(* CODESYS project Pistons innlevering 4 Biraveen.export

Project tree, tasks and I/O mapping:
  Device : CODESYS Control Win V3 x64, 3S - Smart Software Solutions GmbH, version 3.5.16.30
    application Application
      libraries: Standard, * (System)
      task MainTask (cyclic, interval 100 ms, priority 1) calls PLC_PRG
      task VISU_TASK (cyclic, interval 100 ms, priority 31) calls VisuElems.Visu_Prg
      global variables GVL
      function block egendefinert_ANDport [ST]
      function block Pistons [ST]
      program PLC_PRG [CFC]
      function block POU [ST]
      function block POU_1 [ST]
      function block seq4 [ST]
      function block Seq_1 [ST]
      visualisation Visualization
*)

// Device/Application/GVL
{attribute 'qualified_only'}
VAR_GLOBAL
	Piston1_IN: BOOL;
	Piston1_OUT: BOOL;
	Piston2_IN: BOOL;
	Piston2_OUT: BOOL;
	Piston3_IN: BOOL;
	Piston3_OUT: BOOL;
	Piston4_IN: BOOL;
	Piston4_OUT: BOOL;
END_VAR

// Device/Application/PLC_PRG
PROGRAM PLC_PRG
VAR
	Pistons_1: Pistons;
	RESET_0: POU; // første sekvens
	Start_knapp: BOOL;
	ElapsedTIme: TIME;
	TON_0: TON;
	DELAY_1: TON;
	Seq_1_0: Seq_1; // andre sekvens
	Delay_2: TON;
	seq_2: POU_1; // tredje sekvens
	Delay_3: TON;
	Seq_3: seq4; //dette er fjerde sekvens
	Delay_4: TON;
	port: egendefinert_ANDport; // egt en OR port-ish!!
	Delay_5: TON; // RESET delayen
END_VAR

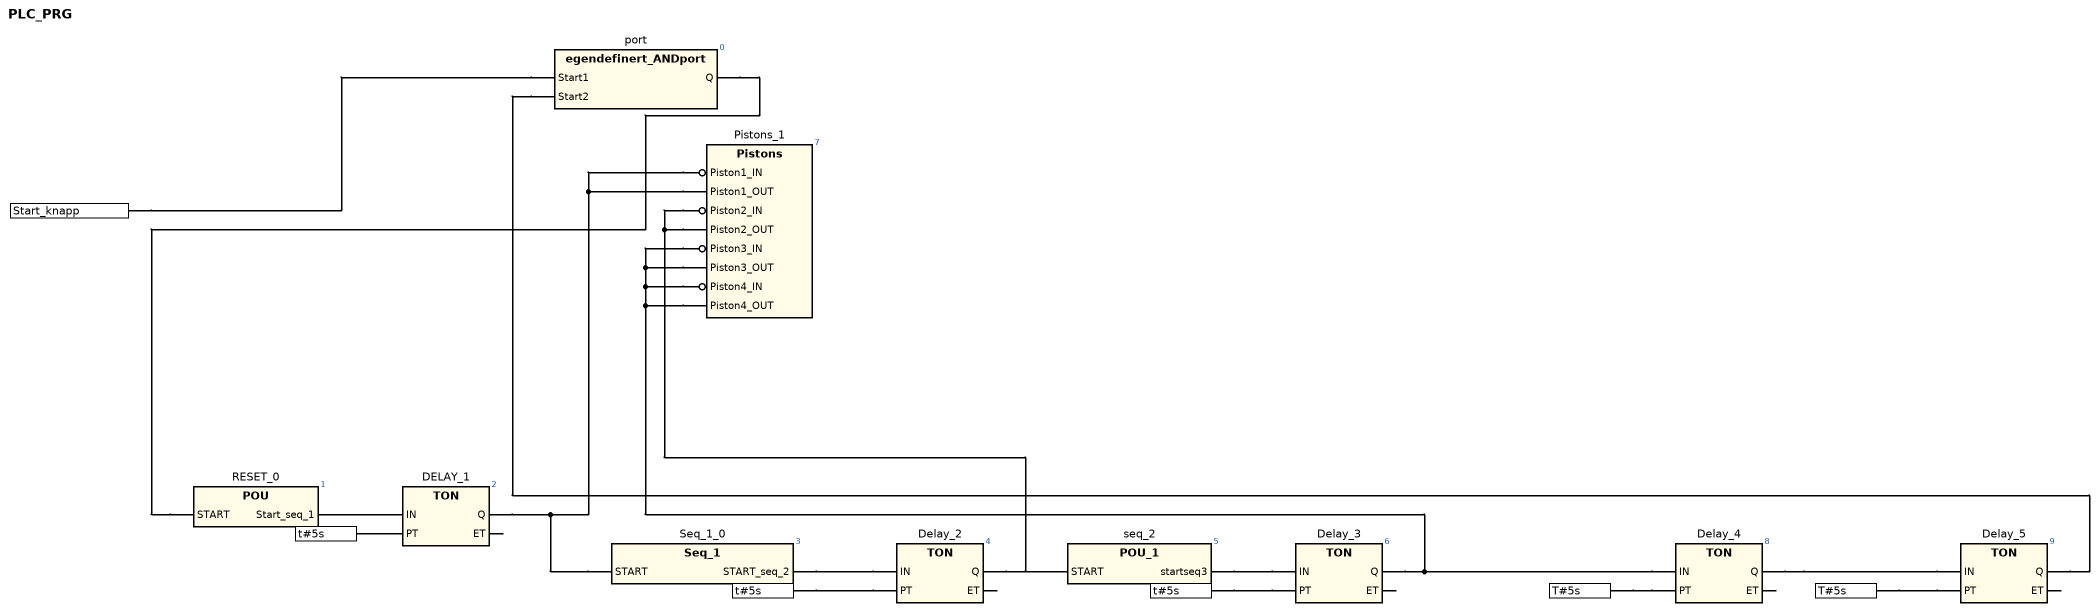
port(Start1 := Start_knapp, Start2 := Delay_5.Q); // egendefinert_ANDport
RESET_0(START := port.Q); // POU
DELAY_1(IN := RESET_0.Start_seq_1, PT := t#5s); // TON
Seq_1_0(START := DELAY_1.Q); // Seq_1
Delay_2(IN := Seq_1_0.START_seq_2, PT := t#5s); // TON
seq_2(START := Delay_2.Q); // POU_1
Delay_3(IN := seq_2.startseq3, PT := t#5s); // TON
Pistons_1(
    Piston1_IN := NOT DELAY_1.Q,
    Piston1_OUT := DELAY_1.Q,
    Piston2_IN := NOT Delay_2.Q,
    Piston2_OUT := Delay_2.Q,
    Piston3_IN := NOT Delay_3.Q,
    Piston3_OUT := Delay_3.Q,
    Piston4_IN := NOT Delay_3.Q,
    Piston4_OUT := Delay_3.Q); // Pistons
Delay_4(IN := Delay_3.Q, PT := T#5s); // TON
Delay_5(IN := Delay_4.Q, PT := T#5s); // TON

END_PROGRAM

// Device/Application/Pistons
FUNCTION_BLOCK Pistons
VAR_INPUT
	Piston1_IN : BOOL := FALSE;
	Piston1_OUT : BOOL := FALSE;
	Piston2_IN : BOOL := FALSE;
	Piston2_OUT : BOOL := FALSE;
	Piston3_IN : BOOL := FALSE;
	Piston3_OUT : BOOL := FALSE;
	Piston4_IN : BOOL := FALSE;
	Piston4_OUT : BOOL := FALSE;

END_VAR
VAR_OUTPUT
END_VAR
VAR
	Hide_Piston_1 : BOOL := TRUE;
	Hide_Piston_2 : BOOL := TRUE;
	Hide_Piston_3 : BOOL := TRUE;
	Hide_Piston_4 : BOOL := TRUE;
	Reset : BOOL := FALSE;
	Start: BOOL;
	Variabel_1: REAL;
	Tstart1 : TIME;
	variabel: REAL;
END_VAR

IF NOT Reset THEN
	
	IF Piston1_OUT AND NOT Piston1_IN THEN 
		Hide_Piston_1 := FALSE;
	ELSIF Piston1_IN AND NOT Piston1_OUT THEN
		Hide_Piston_1 := TRUE;
	ELSE
		Hide_Piston_1 := Hide_Piston_1;
	END_IF

	IF Piston2_OUT AND NOT Piston2_IN THEN
		Hide_Piston_2 := FALSE;
	ELSIF Piston2_IN AND NOT Piston2_OUT THEN
		Hide_Piston_2 := TRUE;
	ELSE
		Hide_Piston_2 := Hide_Piston_2;
	END_IF

	IF Piston3_OUT AND NOT Piston3_IN THEN
		Hide_Piston_3 := FALSE;
	ELSIF Piston3_IN AND NOT Piston3_OUT THEN
		Hide_Piston_3 := TRUE;
	ELSE
		Hide_Piston_3 := Hide_Piston_3;
	END_IF
	
	IF Piston4_OUT AND NOT Piston4_IN THEN
		Hide_Piston_4 := FALSE;
	ELSIF Piston4_IN AND NOT Piston4_OUT THEN
		Hide_Piston_4 := TRUE;
	ELSE
		Hide_Piston_4 := Hide_Piston_4;
	END_IF

ELSE
	Hide_Piston_1 := TRUE;
	Hide_Piston_2 := TRUE;
	Hide_Piston_3 := TRUE;
	Hide_Piston_4 := TRUE;
	Piston1_IN := FALSE;
	Piston1_OUT := FALSE;
	Piston2_IN := FALSE;
	Piston2_OUT := FALSE;
	Piston3_IN := FALSE;
	Piston3_OUT := FALSE;
	Piston4_IN := FALSE;
	Piston4_OUT := FALSE;
	variabel := 0;
END_IF

IF Hide_piston_2 = FALSE AND variabel = 0  THEN 
	HIDE_Piston_1 := TRUE;
END_IF

IF Hide_piston_3 = FALSE THEN 
	HIDE_Piston_2 := TRUE;
END_IF

//IF Hide_piston_4 = FALSE THEN 
	//HIDE_Piston_3 := TRUE;
	//variabel := 1;
//END_IF

// IF Hide_piston_4 = FALSE AND variabel = 1 THEN 
	//HIDE_Piston_1 := TRUE;
	//variabel := 0;
//END_IF

END_FUNCTION_BLOCK

// Device/Application/egendefinert_ANDport
FUNCTION_BLOCK egendefinert_ANDport
VAR_INPUT
	Start1 : BOOL;
	Start2 : BOOL;
END_VAR
VAR_OUTPUT
END_VAR
VAR
	Q : BOOL;
END_VAR

IF Start1 = FALSE AND Start2 = FALSE THEN
	Q := FALSE; 
END_IF

IF Start1 = TRUE AND Start2 = FALSE THEN
	Q := TRUE; 
END_IF

IF Start1 = FALSE AND Start2 = TRUE THEN
	Q := TRUE; 
END_IF

IF Start1 = TRUE AND Start2 = TRUE THEN
	Q := FALSE; 
END_IF

IF Q = FALSE AND START2 = TRUE THEN
	Q := TRUE; 
END_IF

END_FUNCTION_BLOCK

// Device/Application/POU_1
FUNCTION_BLOCK POU_1
VAR_INPUT
	START : BOOL;
END_VAR
VAR_OUTPUT
END_VAR
VAR
	Startseq3 : BOOL;
END_VAR

IF START = TRUE THEN 
	STARTseq3 := TRUE;
END_IF

IF START = FALSE THEN 
	STARTseq3 := FALSE;
END_IF

END_FUNCTION_BLOCK

// Device/Application/POU
FUNCTION_BLOCK POU
VAR_INPUT
	START : BOOL;
END_VAR
VAR_OUTPUT

END_VAR
VAR
	Start_seq_1: BOOL;
	pistonin : BOOL;
	pistonut : BOOL;
	wait: TON;
END_VAR


IF START = FALSE THEN
	Start_seq_1 := TRUE;
	Pistonin := TRUE;
	
END_IF

IF START = TRUE THEN 
	Start_seq_1 := FALSE;
END_IF

END_FUNCTION_BLOCK

// Device/Application/Seq_1
FUNCTION_BLOCK Seq_1
VAR_INPUT
	START : BOOL;
END_VAR
VAR_OUTPUT
END_VAR
VAR
	START_seq_2: BOOL;
END_VAR

IF START = TRUE THEN 
	START_seq_2 := TRUE;
END_IF

IF START = FALSE THEN 
	START_seq_2 := FALSE;
END_IF

END_FUNCTION_BLOCK

// Device/Application/seq4
FUNCTION_BLOCK seq4
VAR_INPUT
	START : BOOL;
END_VAR
VAR_OUTPUT
END_VAR
VAR
	Startseq4 : BOOL;
END_VAR

IF START = TRUE THEN 
	STARTseq4 := TRUE;
END_IF

IF START = FALSE THEN 
	STARTseq4 := FALSE;
END_IF

END_FUNCTION_BLOCK

// Device/Application/Visualization
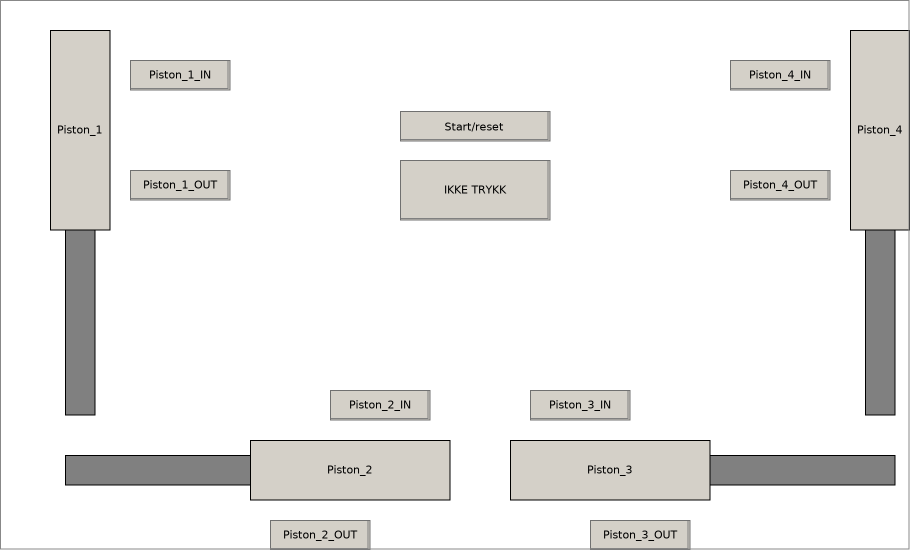
VISUALIZATION Visualization  // 910x550
    Rectangle (865,50 30x200)
    Rectangle (530,455 200x30)
    Rectangle (230,455 200x30)
    Rectangle (65,50 30x200)
    Rectangle (65,215 30x200), invisible if: PLC_PRG.Pistons_1.Hide_Piston_1
    Rectangle (65,455 200x30), invisible if: PLC_PRG.Pistons_1.Hide_Piston_2
    Rectangle (865,215 30x200), invisible if: PLC_PRG.Pistons_1.Hide_Piston_4
    Rectangle (695,455 200x30), invisible if: PLC_PRG.Pistons_1.Hide_Piston_3
    Rectangle (850,30 60x200), "Piston_4"
    Rectangle (50,30 60x200), "Piston_1"
    Rectangle (250,440 200x60), "Piston_2"
    Rectangle (510,440 200x60), "Piston_3"
    Button (400,160 150x60), "IKKE TRYKK"
        tap PLC_PRG.Pistons_1.Reset
    Button (130,170 100x30), "Piston_1_OUT"
        toggle PLC_PRG.Pistons_1.Piston1_OUT p2164770859=TRUE
    Button (130,60 100x30), "Piston_1_IN"
        toggle PLC_PRG.Pistons_1.Piston1_IN
    Button (730,60 100x30), "Piston_4_IN"
        toggle PLC_PRG.Pistons_1.Piston4_IN
    Button (730,170 100x30), "Piston_4_OUT"
        toggle PLC_PRG.Pistons_1.Piston4_OUT
    Button (330,390 100x30), "Piston_2_IN"
        toggle PLC_PRG.Pistons_1.Piston2_IN
    Button (270,520 100x30), "Piston_2_OUT"
        toggle PLC_PRG.Pistons_1.Piston2_OUT
    Button (590,520 100x30), "Piston_3_OUT"
        toggle PLC_PRG.Pistons_1.Piston3_OUT
    Button (530,390 100x30), "Piston_3_IN"
        toggle PLC_PRG.Pistons_1.Piston3_IN
    Button (400,111 150x30)
        toggle PLC_PRG.Start_knapp
    Label (399,112 150x30), "Start/reset"
END_VISUALIZATION
